PROGRAM MAIN
VAR
	fb_child : FB_Child;
END_VAR

END_PROGRAM

(* stored: Version 1.1.0.1, ProductVersion 3.1.4024.12
   POU MAIN: Id {902b5c23-cd84-49c7-9aa7-babb6f1d9b2f}, SpecialFunc None *)
